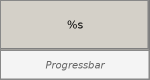
VISUALIZATION UserControlButton  // 150x80
VAR_IN_OUT
	bExecute : BOOL;
	Counter : UDINT;
	sName : STRING;
END_VAR
    Button (0,0 150x50), "%s", text variable: sName
        tap bExecute
        OnMouseDown: execute {  }
    Progressbar (0,50 150x30), variable: Counter
END_VISUALIZATION

(* stored: Version 1.1.0.1, ProductVersion 3.1.4024.12
   Visu UserControlButton: Id {17cef138-b80a-40d5-ac8b-2cff87a93508} *)
